// TIA Portal V17 export
// export: Created 2025-03-10T13:13:17.327371Z, ExportSetting WithDefaults, DisplayName Totally Integrated Automation Portal, DisplayVersion V17 Update 8, DisplayName TIA Portal Openness, DisplayVersion V17 Update 8, DisplayName TIA Portal Version Control Interface, DisplayVersion V17, DisplayName SINAMICS Startdrive Advanced, DisplayVersion V17 SP2, DisplayName SINAMICS Startdrive G110M, G120, G120C, G120D, G120P, G115D, DisplayVersion V17 SP2, DisplayName SINAMICS Startdrive G130, G150, S120, S150, SINAMICS MV, S210, DisplayVersion V17 SP2, DisplayName STEP 7 Professional, DisplayVersion V17 Update 8, DisplayName SINUMERIK ONE STEP 7 Toolbox, DisplayVersion V17 Update 12, DisplayName SINUMERIK 840D sl STEP 7 Toolbox, DisplayVersion V17 Update 12, DisplayName STEP 7 Safety, DisplayVersion V17 Update 6, DisplayName WinCC Advanced, DisplayVersion V17 Update 8
VAR_GLOBAL   // PLC tag table "TAGS_IO_HOPPERS_CLADDING"
   "//////////_HOPPERS_POWDER_FLOW_SENSORS_//////////" AT %M580.0 : Bool;
   "//////////_HOPPERS_WEIGHT_CONTROL_SENSORS_//////////" AT %M596.0 : Bool;
   "/////_HOPPER_JACKET_TEMPERATURE_CONTROL_/////" AT %M150.0 : Bool;   // /////_HOPPER_JACKET_TEMPERATURE_CONTROL/////
   "/////_HOPPER_LEVEL_SENSORS_/////" AT %M70.0 : Bool;   // /////_HOPPER_LEVEL_SENSORS_/////
   "/////_HOPPER_PRESSURE_SENSORS/////" AT %M510.0 : Bool;   // /////_HOPPER_PRESSURE_SENSORS/////
   "/////_HOPPERS_PRESSURE_CONTROLS_/////" AT %M160.0 : Bool;
   "/////_HOPPERS_VALVES_/////" AT %M75.0 : Bool;   // /////_HOPPERS_VALVES_/////
   HPPR_1_MOTOR_ENABLE_1 AT %Q140.4 : Bool;   // HOPPER 1 MOTOR ENABLE SIGNAL 1
   HPPR_1_MOTOR_ENABLE_2 AT %Q140.5 : Bool;   // HOPPER 1 MOTOR ENABLE SIGNAL 2
   HPPR_2_MOTOR_ENABLE_1 AT %Q140.6 : Bool;   // HOPPER 2 MOTOR ENABLE SIGNAL 1
   HPPR_2_MOTOR_ENABLE_2 AT %Q140.7 : Bool;   // HOPPER 2 MOTOR ENABLE SIGNAL 2
   HPPR_3_MOTOR_ENABLE_1 AT %Q142.2 : Bool;   // HOPPER 3 MOTOR ENABLE SIGNAL 1
   HPPR_3_MOTOR_ENABLE_2 AT %Q142.3 : Bool;   // HOPPER 3 MOTOR ENABLE SIGNAL 2
   HPPR_4_MOTOR_ENABLE_1 AT %Q142.4 : Bool;   // HOPPER 4 MOTOR ENABLE SIGNAL 1
   HPPR_4_MOTOR_ENABLE_2 AT %Q142.5 : Bool;   // HOPPER 4 MOTOR ENABLE SIGNAL 2
   HPPR_5_MOTOR_ENABLE_1 AT %Q142.6 : Bool;   // HOPPER 5 MOTOR ENABLE SIGNAL 1
   HPPR_5_MOTOR_ENABLE_2 AT %Q142.7 : Bool;   // HOPPER 5 MOTOR ENABLE SIGNAL 2
   U01_HOPPER_1_HIGH_LEVEL_SENSOR_I AT %I70.1 : Bool;   // UNIT 01 HOPPER 1 HIGH LEVEL SENSOR INPUT
   U01_HOPPER_1_LOW_LEVEL_SENSOR_I AT %I70.0 : Bool;   // UNIT 01 HOPPER 1 LOW LEVEL SENSOR INPUT
   U01_HOPPER_1_LOWER_JACKET_TEMP_CONTROL_I AT %MW162 : Word;   // UNIT 01 HOPPER 1 LOWER JACKET TEMPERATURE CONTROL INPUT
   U01_HOPPER_1_LOWER_JACKET_TEMP_CONTROL_Q AT %MW166 : Word;   // UNIT 01 HOPPER 1 LOWER JACKET TEMPERATURE CONTROL OUTPUT
   U01_HOPPER_1_POWDER_FLOW_SENSOR_I AT %IW580 : Word;   // UNIT 01 HOPPER 1 POWDER FLOW SENSOR INPUT
   U01_HOPPER_1_PRESSURE_SENSOR_I AT %IW510 : Word;   // UNIT 01HOPPER 1 PRESSURE SENSOR INPUT
   U01_HOPPER_1_UPPER_JACKET_TEMP_CONTROL_I AT %MW150 : Word;   // UNIT 01 HOPPER 1 UPPER JACKET TEMPERATURE CONTROL INPUT
   U01_HOPPER_1_UPPER_JACKET_TEMP_CONTROL_Q AT %MW155 : Word;   // UNIT 01 HOPPER 1 UPPER JACKET TEMPERATURE CONTROL OUTPUT
   U01_HOPPER_1_WEIGHT_SENSOR_I AT %IW596 : Word;   // UNIT 01 HOPPER 1 WEIGHT SENSOR INPUT
   U01_HOPPER_2_HIGH_LEVEL_SENSOR_I AT %I70.3 : Bool;   // UNIT 01 HOPPER 2 HIGH LEVEL SENSOR INPUT
   U01_HOPPER_2_LOW_LEVEL_SENSOR_I AT %I70.2 : Bool;   // UNIT 01 HOPPER 2 LOW LEVEL SENSOR INPUT
   U01_HOPPER_2_LOWER_JACKET_TEMP_CONTROL_I AT %MW168 : Word;   // UNIT 01 HOPPER 2 LOWER JACKET TEMPERATURE CONTROL INPUT
   U01_HOPPER_2_LOWER_JACKET_TEMP_CONTROL_Q AT %MW172 : Word;   // UNIT 01 HOPPER 2 LOWER JACKET TEMPERATURE CONTROL OUTPUT
   U01_HOPPER_2_POWDER_FLOW_SENSOR_I AT %IW582 : Word;   // UNIT 01 HOPPER 2 POWDER FLOW SENSOR INPUT
   U01_HOPPER_2_PRESSURE_SENSOR_I AT %IW518 : Word;   // UNIT 01HOPPER 2 PRESSURE SENSOR INPUT
   U01_HOPPER_2_UPPER_JACKET_TEMP_CONTROL_I AT %MW151 : Word;   // UNIT 01 HOPPER 2 UPPER JACKET TEMPERATURE CONTROL INPUT
   U01_HOPPER_2_UPPER_JACKET_TEMP_CONTROL_Q AT %MW156 : Word;   // UNIT 01 HOPPER 2 UPPER JACKET TEMPERATURE CONTROL OUTPUT
   U01_HOPPER_2_WEIGHT_SENSOR_I AT %IW598 : Word;   // UNIT 01 HOPPER 2 WEIGHT SENSOR INPUT
   U01_HPPR_1_CLEANING_VALVE_Q AT %M73.5 : Bool;   // UNIT 01 HOPPER 1 CLEANING VALVE OUTPUT
   U01_HPPR_1_FEEDBACK_PRESSURE_CONTROL_I AT %IW160 : Int;   // UNIT 01 HOPPER 1 FEEDBACK PRESSURE CONTROL INPUT
   U01_HPPR_1_PRESSURE_CONTROL_Q AT %QW160 : Int;   // UNIT 01 HOPPER 1 PRESSURE CONTROL OUTPUT
   U01_HPPR_1_PRESSURIZE_GAS_VALVE_Q AT %Q70.0 : Bool;   // UNIT 01 HOPPER 1 PRESSURIZE GAS VALVE OUTPUT
   U01_HPPR_1_RELIEF_GAS_VALVE_Q AT %Q70.1 : Bool;   // UNIT 01 HOPPER 1 RELIEF GAS VALVE OUTPUT
   U01_HPPR_1_TRANSF_POWDER_VALVE_Q AT %M1500.0 : Bool;   // UNIT 01 HOPPER 1 TRANSFER POWDER VALVE OUTPUT
   U01_HPPR_2_CLEANING_VALVE_Q AT %M73.6 : Bool;   // UNIT 01 HOPPER 2 CLEANING VALVE OUTPUT
   U01_HPPR_2_FEEDBACK_PRESSURE_CONTROL_I AT %IW162 : Int;   // UNIT 01 HOPPER 2 FEEDBACK PRESSURE CONTROL INPUT
   U01_HPPR_2_PRESSURE_CONTROL_Q AT %QW162 : Int;   // UNIT 01 HOPPER 2 PRESSURE CONTROL OUTPUT
   U01_HPPR_2_PRESSURIZE_GAS_VALVE_Q AT %Q70.2 : Bool;   // UNIT 01 HOPPER 2 PRESSURIZE GAS VALVE OUTPUT
   U01_HPPR_2_RELIEF_GAS_VALVE_Q AT %Q70.3 : Bool;   // UNIT 01 HOPPER 2 RELIEF GAS VALVE OUTPUT
   U01_HPPR_2_TRANSF_POWDER_VALVE_Q AT %M1500.1 : Bool;   // UNIT 01 HOPPER 2 TRANSFER POWDER VALVE OUTPUT
   U02_HOPPER_1_HIGH_LEVEL_SENSOR_I AT %I70.5 : Bool;   // UNIT 02 HOPPER 1 HIGH LEVEL SENSOR INPUT
   U02_HOPPER_1_LOW_LEVEL_SENSOR_I AT %I70.4 : Bool;   // UNIT 02 HOPPER 1 LOW LEVEL SENSOR INPUT
   U02_HOPPER_1_LOWER_JACKET_TEMP_CONTROL_I AT %MW176 : Word;   // UNIT 02 HOPPER 1 LOWER JACKET TEMPERATURE CONTROL INPUT
   U02_HOPPER_1_LOWER_JACKET_TEMP_CONTROL_Q AT %MW178 : Word;   // UNIT 02 HOPPER 1 LOWER JACKET TEMPERATURE CONTROL OUTPUT
   U02_HOPPER_1_POWDER_FLOW_SENSOR_I AT %IW584 : Word;   // UNIT 02 HOPPER 1 POWDER FLOW SENSOR INPUT
   U02_HOPPER_1_PRESSURE_SENSOR_I AT %IW526 : Word;   // UNIT 02 HOPPER 1 PRESSURE SENSOR INPUT
   U02_HOPPER_1_UPPER_JACKET_TEMP_CONTROL_I AT %MW152 : Word;   // UNIT 02 HOPPER 1 UPPER JACKET TEMPERATURE CONTROL INPUT
   U02_HOPPER_1_UPPER_JACKET_TEMP_CONTROL_Q AT %MW157 : Word;   // UNIT 02 HOPPER 1 UPPER JACKET TEMPERATURE CONTROL OUTPUT
   U02_HOPPER_1_WEIGHT_SENSOR_I AT %IW600 : Word;   // UNIT 02 HOPPER 1 WEIGHT SENSOR INPUT
   U02_HOPPER_2_HIGH_LEVEL_SENSOR_I AT %I70.7 : Bool;   // UNIT 02 HOPPER 2 HIGH LEVEL SENSOR INPUT
   U02_HOPPER_2_LOW_LEVEL_SENSOR_I AT %I70.6 : Bool;   // UNIT 02 HOPPER 2 LOW LEVEL SENSOR INPUT
   U02_HOPPER_2_LOWER_JACKET_TEMP_CONTROL_I AT %MW164 : Word;   // UNIT 02 HOPPER 2 LOWER JACKET TEMPERATURE CONTROL INPUT
   U02_HOPPER_2_LOWER_JACKET_TEMP_CONTROL_Q AT %MW174 : Word;   // UNIT 02 HOPPER 2 LOWER JACKET TEMPERATURE CONTROL OUTPUT
   U02_HOPPER_2_POWDER_FLOW_SENSOR_I AT %IW588 : Word;   // UNIT 02 HOPPER 2 POWDER FLOW SENSOR INPUT
   U02_HOPPER_2_PRESSURE_SENSOR_I AT %IW534 : Word;   // UNIT 02 HOPPER 2 PRESSURE SENSOR INPUT
   U02_HOPPER_2_UPPER_JACKET_TEMP_CONTROL_I AT %MW153 : Word;   // UNIT 02 HOPPER 2 UPPER JACKET TEMPERATURE CONTROL INPUT
   U02_HOPPER_2_UPPER_JACKET_TEMP_CONTROL_Q AT %MW158 : Word;   // UNIT 02 HOPPER 2 UPPER JACKET TEMPERATURE CONTROL OUTPUT
   U02_HOPPER_2_WEIGHT_SENSOR_I AT %IW602 : Word;   // UNIT 02 HOPPER 2 WEIGHT SENSOR INPUT
   U02_HOPPER_3_HIGH_LEVEL_SENSOR_I AT %I71.1 : Bool;   // UNIT 02 HOPPER 3 HIGH LEVEL SENSOR INPUT
   U02_HOPPER_3_LOW_LEVEL_SENSOR_I AT %I71.0 : Bool;   // UNIT 02 HOPPER 3 LOW LEVEL SENSOR INPUT
   U02_HOPPER_3_LOWER_JACKET_TEMP_CONTROL_I AT %MW170 : Word;   // UNIT 02 HOPPER 3 LOWER JACKET TEMPERATURE CONTROL INPUT
   U02_HOPPER_3_LOWER_JACKET_TEMP_CONTROL_Q AT %MW180 : Word;   // UNIT 02 HOPPER 3 LOWER JACKET TEMPERATURE CONTROL OUTPUT
   U02_HOPPER_3_POWDER_FLOW_SENSOR_I AT %IW590 : Word;   // UNIT 02 HOPPER 3 POWDER FLOW SENSOR INPUT
   U02_HOPPER_3_PRESSURE_SENSOR_I AT %IW542 : Word;   // UNIT 02 HOPPER 3 PRESSURE SENSOR INPUT
   U02_HOPPER_3_UPPER_JACKET_TEMP_CONTROL_I AT %MW154 : Word;   // UNIT 02 HOPPER 3 UPPER JACKET TEMPERATURE CONTROL INPUT
   U02_HOPPER_3_UPPER_JACKET_TEMP_CONTROL_Q AT %MW159 : Word;   // UNIT 02 HOPPER 3 UPPER JACKET TEMPERATURE CONTROL OUTPUT
   U02_HOPPER_3_WEIGHT_SENSOR_I AT %IW586 : Word;   // UNIT 02 HOPPER 3 WEIGHT SENSOR INPUT
   U02_HPPR_1_CLEANING_VALVE_Q AT %M73.7 : Bool;   // UNIT 02 HOPPER 1 CLEANING VALVE OUTPUT
   U02_HPPR_1_FEEDBACK_PRESSURE_CONTROL_I AT %IW164 : Int;   // UNIT 02 HOPPER 1 FEEDBACK PRESSURE CONTROL INPUT
   U02_HPPR_1_PRESSURE_CONTROL_Q AT %QW164 : Int;   // UNIT 02 HOPPER 1 PRESSURE CONTROL OUTPUT
   U02_HPPR_1_PRESSURIZE_GAS_VALVE_Q AT %Q70.4 : Bool;   // UNIT 02 HOPPER 1 PRESSURIZE GAS VALVE OUTPUT
   U02_HPPR_1_RELIEF_GAS_VALVE_Q AT %Q70.5 : Bool;   // UNIT 02 HOPPER 1 RELIEF GAS VALVE OUTPUT
   U02_HPPR_1_TRANSF_POWDER_VALVE_Q AT %M1500.2 : Bool;   // UNIT 02 HOPPER 1 TRANSFER POWDER VALVE OUTPUT
   U02_HPPR_2_CLEANING_VALVE_Q AT %M74.0 : Bool;   // UNIT 02 HOPPER 2 CLEANING VALVE OUTPUT
   U02_HPPR_2_FEEDBACK_PRESSURE_CONTROL_I AT %IW166 : Int;   // UNIT 02 HOPPER 2 FEEDBACK PRESSURE CONTROL INPUT
   U02_HPPR_2_PRESSURE_CONTROL_Q AT %QW166 : Int;   // UNIT 02 HOPPER 2 PRESSURE CONTROL OUTPUT
   U02_HPPR_2_PRESSURIZE_GAS_VALVE_Q AT %Q70.6 : Bool;   // UNIT 02 HOPPER 2 PRESSURIZE GAS VALVE OUTPUT
   U02_HPPR_2_RELIEF_GAS_VALVE_Q AT %Q70.7 : Bool;   // UNIT 02 HOPPER 2 RELIEF GAS VALVE OUTPUT
   U02_HPPR_2_TRANSF_POWDER_VALVE_Q AT %M1500.3 : Bool;   // UNIT 02 HOPPER 2 TRANSFER POWDER VALVE OUTPUT
   U02_HPPR_3_CLEANING_VALVE_Q AT %M1500.5 : Bool;   // UNIT 02 HOPPER 3 CLEANING VALVE OUTPUT
   U02_HPPR_3_FEEDBACK_PRESSURE_CONTROL_I AT %IW168 : Int;   // UNIT 02 HOPPER 3 FEEDBACK PRESSURE CONTROL INPUT
   U02_HPPR_3_PRESSURE_CONTROL_Q AT %QW170 : Int;   // UNIT 02 HOPPER 3 PRESSURE CONTROL OUTPUT
   U02_HPPR_3_PRESSURIZE_GAS_VALVE_Q AT %Q71.0 : Bool;   // UNIT 02 HOPPER 3 PRESSURIZE GAS VALVE OUTPUT
   U02_HPPR_3_RELIEF_GAS_VALVE_Q AT %Q71.1 : Bool;   // UNIT 02 HOPPER 3 RELIEF GAS VALVE OUTPUT
   U02_HPPR_3_TRANSF_POWDER_VALVE_Q AT %M1500.4 : Bool;   // UNIT 02 HOPPER 3 TRANSFER POWDER VALVE OUTPUT
END_VAR
